// TIA Portal V19 export
TYPE "IF_Commands"
   STRUCT
      Commando_1 : Bool;   // (1) Upload Start
      Commando_2 : Bool;   // (2) Upload End
      Commando_3 : Bool;   // (3) Download Start
      Commando_4 : Bool;   // (4) Download End
      Commando_5 : Bool;   // (5) Store
      Commando_6 : Bool;   // (6) Break
      Commando_7 : Bool;   // (130) Restore Factory Settings
      Commando_8 : Bool;   // (240) Test Event 8DFE appears
      Commando_9 : Bool;   // (241) Test Event 8DFE disappears
      Commando_10 : Bool;   // (242) Test Event 8DFF appears
      Commando_11 : Bool;   // (243) Test Event 8DFF disappears
      Commando_12 : Bool;   // not used
      Commando_13 : Bool;   // not used
      Commando_14 : Bool;   // not used
      Commando_15 : Bool;   // not used
      Commando_16 : Bool;   // not used
      Commando_17 : Bool;   // not used
      Commando_18 : Bool;   // not used
      Commando_19 : Bool;   // not used
      Commando_20 : Bool;   // not used
      Commando_21 : Bool;   // not used
      Commando_22 : Bool;   // not used
      Commando_23 : Bool;   // not used
      Commando_24 : Bool;   // not used
   END_STRUCT;
END_TYPE
